FUNCTION_BLOCK Test_TStreamAdd_Read_ULINT EXTENDS T_UnitTestBase
VAR
    Stream  : T_Stream(StreamLength := 2);
    ArgType : E_ArgTypeId := E_ArgTypeId.Type_ULINT;
END_VAR


Stream.Init(2);

// add a ULINT...
Stream.SetNextArgTypeId(ArgType);
Stream.Add_ULINT(123456789);

Stream.SetReadPosition(0);

// check next arg type is correct...
Assertion.AssertEquals_INT(Expected     := ArgType,
                           Actual       := Stream.GetNextArgTypeId(),
                           VariableName := 'Stream.GetNextArgTypeId()');

// check next value...	
Assertion.AssertEquals_ULINT(Expected     := 123456789,
                             Actual       := Stream.Read_ULINT(),
                             VariableName := 'Stream.Read_ULINT()');

// check we are at the end of the stream..							
Assertion.AssertEquals_UDINT(Expected     := Stream.StreamLength,
                             Actual       := Stream.ReadPosition,
                             VariableName := 'Stream.ReadPosition');

TestFinished();

END_FUNCTION_BLOCK

(* stored: Version 1.1.0.1, ProductVersion 3.1.4024.9
   POU Test_TStreamAdd_Read_ULINT: Id {5e9ca6f8-35eb-48c2-9787-f5c46dfb8761}, SpecialFunc None *)
